// TIA Portal V19 export
FUNCTION_BLOCK "MatLub_Count_FB"   // FB156, LAD
TITLE = MATERIAL LUBRICATION (ROLL)
// stored: MemoryReserve 100, SetENOAutomatically false
   VAR_INPUT
      AreaInterface : "AreaInterface";
      DataIn : Struct
         PbStop : Bool;
         PbStart : Bool;
         SensorLevel : Bool;
         PumpFeedbackRunning : Bool;
      END_STRUCT;
      CIn : Struct
         EnableStopInPhase : Bool;
         EnableStopProgrammed : Bool;
         MaterialCounter : LReal;
      END_STRUCT;
      Config : Struct
         EnableWngSystemOff : Bool;
         LowTankLevelDly : Time;
      END_STRUCT;
   END_VAR
   VAR_OUTPUT
      MachineInterface : "MachineInterface";
      DataOut : Struct
         M_Pump_Contactor : Bool;
         Lamp : Bool;
      END_STRUCT;
      COut : Struct
         PumpIsRunning : Bool;
      END_STRUCT;
   END_VAR
   VAR_IN_OUT
      PersistentValues : Struct
         Par : Struct
            Enable : Bool;
            OnDuration : Time;
            SpaceInterval : LReal;
         END_STRUCT;
      END_STRUCT;
   END_VAR
   VAR
      Sts : Struct
         AlarmsPresence : Bool;
         WarningsPresence : Bool;
         IsStandstill : Bool;
         PumpRunReq : Bool;
         LastFeed : LReal;
         PrevMatcounter : LReal;
         MaterialFed : LReal;
         Pump_Cnd { ExternalAccessible := 'False'; ExternalVisible := 'False'; ExternalWritable := 'False'} : Bool;
         Blower_Cnd { ExternalAccessible := 'False'; ExternalVisible := 'False'; ExternalWritable := 'False'} : Bool;
         Cloth_Cnd { ExternalAccessible := 'False'; ExternalVisible := 'False'; ExternalWritable := 'False'} : Bool;
      END_STRUCT;
      Ctrl : Struct
         RstAlarms : Bool;
         StopInPhase : Bool;
         StopProgrammed : Bool;
         Pump_ManStart : Bool;
         Pump_AutStart : Bool;
         Blower_ManStart : Bool;
         Blower_AutStart : Bool;
         Cloth_AutStart : Bool;
      END_STRUCT;
      Alr : Struct
         LowTankLevel : Bool;
         MPump : "MotorAlr";
      END_STRUCT;
      Wng : Struct
         NoAutReady : Bool;
         PumpOff : Bool;
      END_STRUCT;
      M_Pump : "Motor";
      TON_DelayBlowerStop { S7_SetPoint := 'True'} : IEC_TIMER;
      TON_DelayPumpStop { S7_SetPoint := 'True'} : IEC_TIMER;
      TON_LowTankLevel { S7_SetPoint := 'True'} : IEC_TIMER;
      Pb_PumpStart_PEAux : Bool;
      Pb_BlowerStart_PEAux : Bool;
   END_VAR
   VAR_TEMP   // added for the SCL form of the ladder/FBD networks
      _w1 : Bool;
   END_VAR
BEGIN

REGION Network 1 (SCL): Reset alarms command
   #Ctrl.RstAlarms := #AreaInterface.RstAlarms;

   IF #Ctrl.RstAlarms THEN
       #Wng.NoAutReady := FALSE;
       #Alr.LowTankLevel := FALSE;
   END_IF;
END_REGION

REGION Network 2: Warning Pump / Blower off
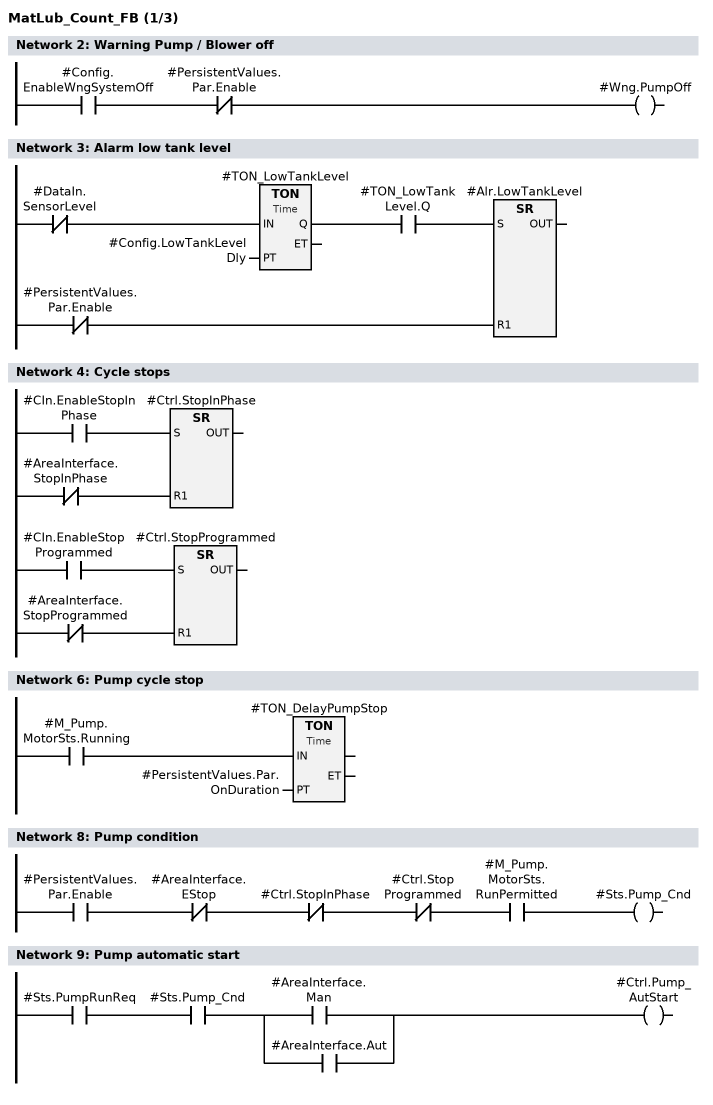
   RUNG wire#powerrail
      Contact( #Config.EnableWngSystemOff )
      I_Contact( #PersistentValues.Par.Enable )
      Coil( #Wng.PumpOff )
   END_RUNG
   // the same network as SCL:
   #Wng.PumpOff := #Config.EnableWngSystemOff AND NOT #PersistentValues.Par.Enable;
END_REGION

REGION Network 3: Alarm low tank level
   RUNG wire#powerrail
      I_Contact( #DataIn.SensorLevel )
      { S7_Templates := "time_type := Time" } #TON_LowTankLevel.TON(pt := #Config.LowTankLevelDly, et =>)
      Contact( #TON_LowTankLevel.Q )
      S_SR(operand := #Alr.LowTankLevel, r1 := wire#w1)
   END_RUNG
   RUNG wire#powerrail
      I_Contact( #PersistentValues.Par.Enable )
   END_RUNG wire#w1
   // the same network as SCL:
   #TON_LowTankLevel.TON(IN := NOT #DataIn.SensorLevel, PT := #Config.LowTankLevelDly);
   IF #TON_LowTankLevel.Q AND #TON_LowTankLevel.Q THEN
       #Alr.LowTankLevel := TRUE;   // SR flip-flop
   END_IF;
   IF NOT #PersistentValues.Par.Enable THEN #Alr.LowTankLevel := FALSE; END_IF;
END_REGION

REGION Network 4: Cycle stops
   RUNG wire#powerrail
      Contact( #CIn.EnableStopInPhase )
      S_SR(operand := #Ctrl.StopInPhase, r1 := wire#w1)
   END_RUNG
   RUNG wire#powerrail
      I_Contact( #AreaInterface.StopInPhase )
   END_RUNG wire#w1
   RUNG wire#powerrail
      Contact( #CIn.EnableStopProgrammed )
      S_SR(operand := #Ctrl.StopProgrammed, r1 := wire#w2)
   END_RUNG
   RUNG wire#powerrail
      I_Contact( #AreaInterface.StopProgrammed )
   END_RUNG wire#w2
   // the same network as SCL:
   IF #CIn.EnableStopInPhase THEN
       #Ctrl.StopInPhase := TRUE;   // SR flip-flop
   END_IF;
   IF NOT #AreaInterface.StopInPhase THEN #Ctrl.StopInPhase := FALSE; END_IF;
   IF #CIn.EnableStopProgrammed THEN
       #Ctrl.StopProgrammed := TRUE;   // SR flip-flop
   END_IF;
   IF NOT #AreaInterface.StopProgrammed THEN #Ctrl.StopProgrammed := FALSE; END_IF;
END_REGION

REGION Network 5: <<< PUMP >>>
END_REGION

REGION Network 6: Pump cycle stop
   RUNG wire#powerrail
      Contact( #M_Pump.MotorSts.Running )
      { S7_Templates := "time_type := Time" } #TON_DelayPumpStop.TON(pt := #PersistentValues.Par.OnDuration, et =>)
   END_RUNG
   // the same network as SCL:
   #TON_DelayPumpStop.TON(IN := #M_Pump.MotorSts.Running, PT := #PersistentValues.Par.OnDuration);
END_REGION

REGION Network 7 (SCL): Pump run request
   #Sts.LastFeed := "M_PosAMinusPosB"(PosA:=#CIn.MaterialCounter,PosB:=#Sts.PrevMatcounter,MODULE := "MATERIAL_COUNTERS_MODULE");
   #Sts.PrevMatcounter := #CIn.MaterialCounter;

   IF #Sts.LastFeed > 1000.0 THEN
       #Sts.LastFeed := 0;
   END_IF;

   #Sts.MaterialFed := #Sts.MaterialFed + #Sts.LastFeed;

   IF  #PersistentValues.Par.OnDuration = T#0s OR #PersistentValues.Par.SpaceInterval <= 0.0 OR NOT #PersistentValues.Par.Enable THEN
       #Sts.PumpRunReq := FALSE;       
   ELSIF   #TON_DelayPumpStop.Q THEN
       #Sts.PumpRunReq := FALSE;   
       #Sts.MaterialFed := 0.0;

   ELSIF NOT #Sts.PumpRunReq AND #Sts.MaterialFed >= #PersistentValues.Par.SpaceInterval THEN
       #Sts.PumpRunReq := true;
   END_IF;
END_REGION

REGION Network 8: Pump condition
   RUNG wire#powerrail
      Contact( #PersistentValues.Par.Enable )
      I_Contact( #AreaInterface.EStop )
      I_Contact( #Ctrl.StopInPhase )
      I_Contact( #Ctrl.StopProgrammed )
      Contact( #M_Pump.MotorSts.RunPermitted )
      Coil( #Sts.Pump_Cnd )
   END_RUNG
   // the same network as SCL:
   #Sts.Pump_Cnd := #PersistentValues.Par.Enable AND NOT #AreaInterface.EStop AND NOT #Ctrl.StopInPhase AND NOT #Ctrl.StopProgrammed AND #M_Pump.MotorSts.RunPermitted;
END_REGION

REGION Network 9: Pump automatic start
   RUNG wire#powerrail
      Contact( #Sts.PumpRunReq )
      Contact( #Sts.Pump_Cnd )
      wire#w1
      Contact( #AreaInterface.Man )
      wire#w2
      Coil( #Ctrl.Pump_AutStart )
   END_RUNG
   RUNG wire#w1
      Contact( #AreaInterface.Aut )
   END_RUNG wire#w2
   // the same network as SCL:
   #Ctrl.Pump_AutStart := #Sts.PumpRunReq AND #Sts.Pump_Cnd AND (#AreaInterface.Man OR #AreaInterface.Aut);
END_REGION

REGION Network 10: Pump manual start
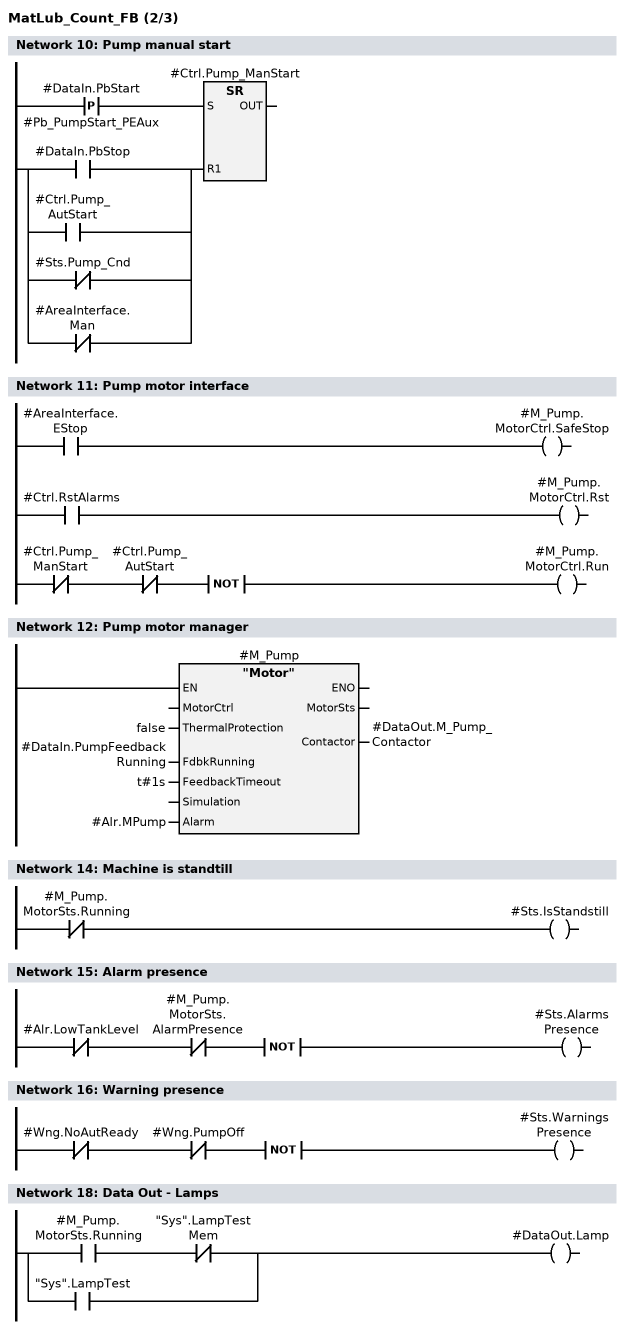
   RUNG wire#powerrail
      P_Contact(operand := #DataIn.PbStart, bit := #Pb_PumpStart_PEAux)
      S_SR(operand := #Ctrl.Pump_ManStart, r1 := wire#w1)
   END_RUNG
   RUNG wire#powerrail
      Contact( #DataIn.PbStop )
   END_RUNG wire#w1
   RUNG wire#powerrail
      Contact( #Ctrl.Pump_AutStart )
   END_RUNG wire#w1
   RUNG wire#powerrail
      I_Contact( #Sts.Pump_Cnd )
   END_RUNG wire#w1
   RUNG wire#powerrail
      I_Contact( #AreaInterface.Man )
   END_RUNG wire#w1
   // the same network as SCL:
   #_w1 := #DataIn.PbStart AND NOT #Pb_PumpStart_PEAux;   // rising edge of #DataIn.PbStart
   #Pb_PumpStart_PEAux := #DataIn.PbStart;
   IF #_w1 THEN
       #Ctrl.Pump_ManStart := TRUE;   // SR flip-flop
   END_IF;
   IF #DataIn.PbStop OR #Ctrl.Pump_AutStart OR NOT #Sts.Pump_Cnd OR NOT #AreaInterface.Man THEN
       #Ctrl.Pump_ManStart := FALSE;
   END_IF;
END_REGION

REGION Network 11: Pump motor interface
   RUNG wire#powerrail
      Contact( #AreaInterface.EStop )
      Coil( #M_Pump.MotorCtrl.SafeStop )
   END_RUNG
   RUNG wire#powerrail
      Contact( #Ctrl.RstAlarms )
      Coil( #M_Pump.MotorCtrl.Rst )
   END_RUNG
   RUNG wire#powerrail
      I_Contact( #Ctrl.Pump_ManStart )
      I_Contact( #Ctrl.Pump_AutStart )
      Not()
      Coil( #M_Pump.MotorCtrl.Run )
   END_RUNG
   // the same network as SCL:
   #M_Pump.MotorCtrl.SafeStop := #AreaInterface.EStop;
   #M_Pump.MotorCtrl.Rst := #Ctrl.RstAlarms;
   #M_Pump.MotorCtrl.Run := NOT (NOT #Ctrl.Pump_ManStart AND NOT #Ctrl.Pump_AutStart);
END_REGION

REGION Network 12: Pump motor manager
   RUNG wire#powerrail
      #M_Pump(MotorCtrl :=, ThermalProtection := false, FdbkRunning := #DataIn.PumpFeedbackRunning, FeedbackTimeout := t#1s, Simulation :=, Alarm := #Alr.MPump, MotorSts =>, Contactor => #DataOut.M_Pump_Contactor)
   END_RUNG
   // the same network as SCL:
   #M_Pump(ThermalProtection := false,   // "Motor"
           FdbkRunning := #DataIn.PumpFeedbackRunning,
           FeedbackTimeout := t#1s,
           Alarm := #Alr.MPump,
           Contactor => #DataOut.M_Pump_Contactor);
END_REGION

REGION Network 13: <<< >>>
END_REGION

REGION Network 14: Machine is standtill
   RUNG wire#powerrail
      I_Contact( #M_Pump.MotorSts.Running )
      Coil( #Sts.IsStandstill )
   END_RUNG
   // the same network as SCL:
   #Sts.IsStandstill := NOT #M_Pump.MotorSts.Running;
END_REGION

REGION Network 15: Alarm presence
   RUNG wire#powerrail
      I_Contact( #Alr.LowTankLevel )
      I_Contact( #M_Pump.MotorSts.AlarmPresence )
      Not()
      Coil( #Sts.AlarmsPresence )
   END_RUNG
   // the same network as SCL:
   #Sts.AlarmsPresence := NOT (NOT #Alr.LowTankLevel AND NOT #M_Pump.MotorSts.AlarmPresence);
END_REGION

REGION Network 16: Warning presence
   RUNG wire#powerrail
      I_Contact( #Wng.NoAutReady )
      I_Contact( #Wng.PumpOff )
      Not()
      Coil( #Sts.WarningsPresence )
   END_RUNG
   // the same network as SCL:
   #Sts.WarningsPresence := NOT (NOT #Wng.NoAutReady AND NOT #Wng.PumpOff);
END_REGION

REGION Network 17 (SCL): Collect machine to area interface
   // Status machine ready
   #MachineInterface.AutReady := #AreaInterface.Aut AND NOT #Sts.AlarmsPresence;
   // Status machine aborting
   #MachineInterface.Aborting := #Sts.AlarmsPresence;
   // Status Ack Stop in phase
   #MachineInterface.AckStopInPhase := #Ctrl.StopInPhase AND #MachineInterface.MotionsStandStill;
   // Status Ack Stop programmed
   #MachineInterface.AckStopProgrammed := #Ctrl.StopProgrammed AND #MachineInterface.MotionsStandStill;
   // Status Motion standtill
   #MachineInterface.MotionsStandStill := #Sts.IsStandstill;
   // Status Alarm presence
   #MachineInterface.AlarmsPresence := #Sts.AlarmsPresence;
   // Status Warning presence
   #MachineInterface.WarningPresence := #Sts.WarningsPresence;

   // Warning machine not automatic ready
   IF #AreaInterface.CheckAutReady AND NOT #MachineInterface.AutReady THEN
     #Wng.NoAutReady := false;
   END_IF;
END_REGION

REGION Network 18: Data Out - Lamps
   RUNG wire#powerrail
      Contact( #M_Pump.MotorSts.Running )
      I_Contact( "Sys".LampTestMem )
      wire#w1
      Coil( #DataOut.Lamp )
   END_RUNG
   RUNG wire#powerrail
      Contact( "Sys".LampTest )
   END_RUNG wire#w1
   // the same network as SCL:
   #DataOut.Lamp := (#M_Pump.MotorSts.Running AND NOT "Sys".LampTestMem) OR "Sys".LampTest;
END_REGION

REGION Network 19: Coordination out
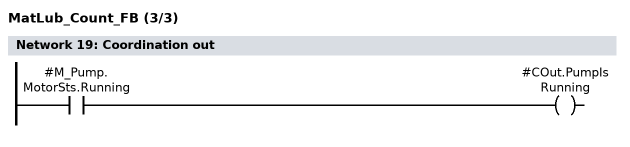
   RUNG wire#powerrail
      Contact( #M_Pump.MotorSts.Running )
      Coil( #COut.PumpIsRunning )
   END_RUNG
   // the same network as SCL:
   #COut.PumpIsRunning := #M_Pump.MotorSts.Running;
END_REGION
END_FUNCTION_BLOCK
